FUNCTION_BLOCK MachineControl
VAR
	_dataService : ITF_MachineDataService;
	MyStatus : INT := 3;
END_VAR

PROPERTY DataService : ITF_MachineDataService
GET
DataService := _dataService;
END_GET
SET
_dataService := DataService;
END_SET
END_PROPERTY

METHOD PushMachineStatus : INT
VAR_INPUT
END_VAR
_dataService.SendStatus(MyStatus);
END_METHOD

END_FUNCTION_BLOCK

(* stored: Version 1.1.0.1, ProductVersion 3.1.4024.12
   POU MachineControl: Id {4b3360ea-25af-4380-9894-e3d9734fb15e}, SpecialFunc None
   Property DataService: Id {1c487fe0-2ce1-4d7c-bdba-697109a49bbf}
   Get Get: Id {7cb3e42e-3129-49ae-9d56-f3c6fa7ca50e}
   Set Set: Id {6e16ea28-19fb-4271-835e-59da4c18f879}
   Method PushMachineStatus: Id {1055d081-0745-4925-8a52-49dc70f23059} *)
